{attribute 'GeneratedUsingTerminal: KL9900-0058'}
{attribute addProperty BoxType "KL9900-0058"}
{attribute addProperty Id "Channel_1AT %Q*Channel_16463F740"}
{attribute addProperty CRC "3483927309"}
{attribute addProperty Size "0"}
TYPE KL_CFA8830D :
STRUCT
	{attribute addProperty Name "Channel_1"}
	Channel_1 : Channel_16463F74;
END_STRUCT
END_TYPE

(* stored: Version 1.2.0.0, ProductVersion 3.1.4024.9
   DUT KL_CFA8830D: Id {84280eb7-be40-4a24-986e-ecd2d458f366} *)
